FUNCTION_BLOCK AR2IO_TO_AR2 (* Composite FB for convert AR2IO to AR2 *)
  (* Standard: 61499-2; Description: Copyright (c) 2024 HR Agrartechnik GmbH This program and the accompanying materials are made available under the terms of the Eclipse Public License 2.0 which is available at https://www.eclipse.org/legal/epl-2.0/ SPDX-License-Identifier: EPL-2.0 *)
  (* Version 1.0, 2024-04-24, Franz Höpfinger, HR Agrartechnik GmbH *)
  PACKAGE adapter::conversion::bidirectional;
  IMPORT eclipse4diac::core::TypeHash;
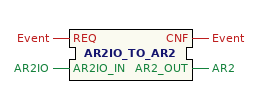
  EVENT_INPUT
    REQ; (* Request to Adapter *)
  END_EVENT
  EVENT_OUTPUT
    CNF; (* Confirmation from Adapter *)
  END_EVENT
  SOCKETS
    AR2IO_IN : adapter::types::bidirectional::AR2IO; (* AR2IO Adapter Input *)
  END_SOCKETS
  PLUGS
    AR2_OUT : adapter::types::bidirectional::AR2; (* AR2 Adapter Output *)
  END_PLUGS
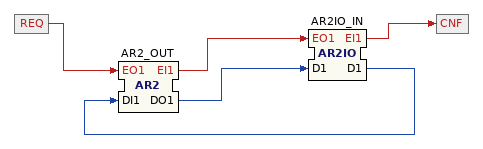
  EVENT_CONNECTIONS
    REQ TO AR2_OUT.EO1;
    AR2IO_IN.EI1 TO CNF;
    AR2_OUT.EI1 TO AR2IO_IN.EO1;
  END_CONNECTIONS
  DATA_CONNECTIONS
    AR2IO_IN.D1 TO AR2_OUT.DI1;
    AR2_OUT.DO1 TO AR2IO_IN.D1;
  END_CONNECTIONS
END_FUNCTION_BLOCK
